FUNCTION_BLOCK FB_HomeAbsoluteSwitch
VAR_INPUT
END_VAR
VAR_OUTPUT
END_VAR
VAR
END_VAR

END_FUNCTION_BLOCK

(* stored: Version 1.1.0.1, ProductVersion 3.1.4022.18
   POU FB_HomeAbsoluteSwitch: Id {4b3b9350-559a-4825-85f8-75f4fbbac869}, SpecialFunc None *)
